{attribute 'qualified_only'}
{attribute 'strict'}
{attribute 'to_string'}
TYPE E_GROUP_CTRL :
(
  GROUP_INVALID,
  GROUP_INIT    := 10,
  GROUP_CLEAR,
  GROUP_BUILD,
  GROUP_ENABLE
)UINT;
END_TYPE

(* stored: Version 1.1.0.1, ProductVersion 3.1.4024.12
   DUT E_GROUP_CTRL: Id {e5fda2d9-7405-444f-8ac0-0f5375b78eeb} *)
